{attribute 'strict'}
TYPE E_CognexCameraGetJobStatus :
(
	WAITING_FOR_STATUS_CODE														:= 2,
	THE_COMMAND_WAS_EXECUTED_SUCCESSFULLY										:= 1,
	UNRECOGNIZED_COMMAND 														:= 0,
	THE_ACTIVE_JOB_HAS_NOT_BEEN_SAVED_OR_DOES_NOT_HAVE_A_NUMERICAL_PREFIX		:= -2
);
END_TYPE

(* stored: Version 1.1.0.1, ProductVersion 3.1.4024.9
   DUT E_CognexCameraGetJobStatus: Id {b4859a11-f9be-43bc-9404-71580ada002c} *)
